TYPE TestStrukturSkill :
STRUCT
	P2P_Movement				:Skill_Position_anfahren; 
	Position					:sRoboterProzessVariablen;
END_STRUCT
END_TYPE

(* stored: Version 1.1.0.1
   DUT TestStrukturSkill: Id {52d9953e-fb64-4002-b191-bc9d8698fb58} *)
